PROGRAM MAIN
VAR
	En:BOOL;
	Shot:BOOL;
	Result:ARRAY [0..7] OF REAL;
END_VAR

Motion.InitMotion();
GVL.Vision();

//Medida temperatura
//MedidaTempPuente();	//Medir la temperatura de los termicos con el puente de resistencias
MedidaTempTarjeta();	//Medir la temperatura de los termicos con la tarjeta EL3202

//ControlTemp();		//Gestion temperatura con bloques TF4110

MedidaDiamMec();	//Medida del diametro con el sensor mecanico

OperatingModes();

IF GVL.Mode = Modes.AUTO THEN
	Basic();
END_IF

Manual();
VisuLogic();
Motion();
GestionVentiladores();

END_PROGRAM

(* stored: Version 1.1.0.1, ProductVersion 3.1.4024.9
   POU MAIN: Id {d8de5791-f153-470a-bfaa-453c619a7f06}, SpecialFunc None *)
